FUNCTION_BLOCK DAerationSensor (* Composite Function Block Type *)
  (* Standard: 61499-2 *)
  (* Version 0.0, 7/1/2024, NVPP, Schneider Electric, template *)
  PACKAGE SE.Nereda;
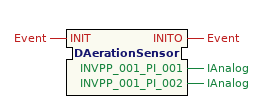
  EVENT_INPUT
    INIT;
  END_EVENT
  EVENT_OUTPUT
    INITO;
  END_EVENT
  PLUGS
    INVPP_001_PI_001 : IAnalog; (* Process value and status interface adapter *)
    INVPP_001_PI_002 : IAnalog; (* Process value and status interface adapter *)
  END_PLUGS
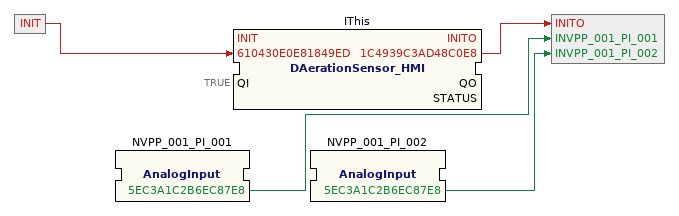
  (* 01 - FUNCTIONNAL INPUT INTERFACE *)
  (* 00 - INITIALIZATION *)
  (* 06 - HMI INTERFACE *)
  (* 02 - FUNCTIONNAL OUTPUT INTERFACE *)
  (* 03 - FIELD INTERFACE *)
  (* Pressure sensor 1 *)
  (* Pressure sensor 2 *)
  FBS
    IThis : DAerationSensor_HMI(QI := TRUE);
    NVPP_001_PI_001 : AnalogInput;
    NVPP_001_PI_002 : AnalogInput;
  END_FBS
  EVENT_CONNECTIONS
    INIT TO IThis.610430E0E81849ED;
    IThis.1C4939C3AD48C0E8 TO INITO;
  END_CONNECTIONS
  ADAPTER_CONNECTIONS
    NVPP_001_PI_001.5EC3A1C2B6EC87E8 TO INVPP_001_PI_001;
    NVPP_001_PI_002.5EC3A1C2B6EC87E8 TO INVPP_001_PI_002;
  END_CONNECTIONS
END_FUNCTION_BLOCK
